{attribute 'qualified_only'}
{attribute 'strict'}
TYPE E_Camera_State :
(
	//GENERIC
	ABORTED				,
	RESET_ERROR			,
	READY				,
	RESET_CMD			,
	//MANUAL_MODE			:=50, /manual mode not needed.
	ERROR				,
	//SPECIFIC FOR EVERY STATION
	HOMING				,
	
	TAKING_PICTURE_PART_PRESENT_INSPECTION	,
	TAKING_PICTURE_CONTINUOUS_PART_PRESENT	,
	TAKING_PICTURE_SEPTUM_POSITION_END		,
	DONE				,
	RESULTS		
);
END_TYPE

(* stored: Version 1.1.0.1, ProductVersion 3.1.4026.18
   DUT E_Camera_State: Id {1f427bb6-b000-49ab-b9fe-b41ba2f3f5a8} *)
